// TIA Portal V20 export
TYPE "LKinCtrl_PointEditor_typePointConfigurationExternalEvents"
// stored: Access Published
   STRUCT
      updatePointTable { ExternalAccessible := 'False'; ExternalVisible := 'False'; ExternalWritable := 'False'} : Bool;
      approachPoint { ExternalAccessible := 'False'; ExternalVisible := 'False'; ExternalWritable := 'False'} : Struct
         trigger : Bool;
         point : "LKinCtrl_typePoint";
      END_STRUCT;
      openTeachKinematics { ExternalAccessible := 'False'; ExternalVisible := 'False'; ExternalWritable := 'False'} : Bool;
   END_STRUCT;
END_TYPE
